// SIMATIC S7-200 project (STEP 7-Micro/WIN), CPU 221 REL 01.10

ORGANIZATION_BLOCK 主程序:OB1
TITLE=程序注释
BEGIN
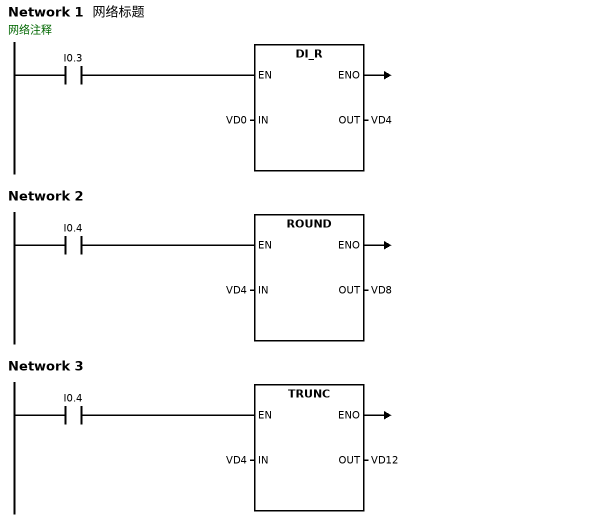
Network 1 // 网络标题
// 网络注释
LD     I0.3
DTR    VD0, VD4
Network 2
LD     I0.4
ROUND  VD4, VD8
Network 3
LD     I0.4
TRUNC  VD4, VD12
END_ORGANIZATION_BLOCK
